FUNCTION_BLOCK ClockInc (* Clock signal generator *)
  (* Standard: 61499-2 *)
  (* Version 1.0, 2008-11-09, Cheng Pang, The University of Auckland, Stable build. *)
  (* Compiler header: package fb.rt.cs725; *)
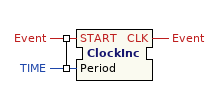
  EVENT_INPUT
    START WITH Period;
  END_EVENT
  EVENT_OUTPUT
    CLK;
  END_EVENT
  VAR_INPUT
    Period : TIME;
  END_VAR
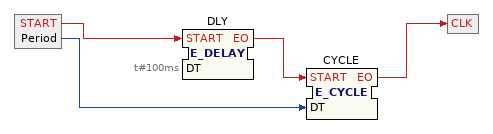
  FBS
    DLY : E_DELAY(DT := t#100ms);
    CYCLE : E_CYCLE;
  END_FBS
  EVENT_CONNECTIONS
    DLY.EO TO CYCLE.START;
    START TO DLY.START;
    CYCLE.EO TO CLK;
  END_CONNECTIONS
  DATA_CONNECTIONS
    Period TO CYCLE.DT;
  END_CONNECTIONS
END_FUNCTION_BLOCK
